// TIA Portal V18 export
VAR_GLOBAL   // PLC tag table "Default tag table"
   Tag_11 AT %M0.0 : Bool;
   Tag_2 AT %M0.1 : Bool;
END_VAR
